FUNCTION TryConvert_STRING_TO_ULINT : BOOL
VAR_INPUT
	in : STRING;
	out : REFERENCE TO ULINT;
END_VAR

IF in <> ULINT_TO_STRING(STRING_TO_ULINT(in)) THEN
	RETURN;
END_IF

out := STRING_TO_ULINT(in);
TryConvert_STRING_TO_ULINT := TRUE;

END_FUNCTION

(* stored: Version 1.1.0.1, ProductVersion 3.1.4024.12
   POU TryConvert_STRING_TO_ULINT: Id {7d016b78-22b5-41ff-b0f5-8e554254e518}, SpecialFunc None *)
